// TIA Portal V19 export
TYPE "LEXCHANGETRAY_typeConstraintRollerEm_toRollerReq"
// stored: Access Published
   STRUCT
      outFeedReq : Bool;   // 请求排料
   END_STRUCT;
END_TYPE
